{attribute 'GeneratedUsingTerminal: EL9930-0000-0017'}
{attribute addProperty BoxType "EL9930-0000-0017"}
{attribute addProperty Id "A_0004_EL9930_0001_0017EL9930_07FC3A1D4"}
{attribute addProperty CRC "2528476189"}
{attribute addProperty Size "4"}
TYPE A_0003_EL9930_0000_0017_96B57C1D EXTENDS EL9930_B8165E3C :
STRUCT
	{attribute addProperty Name "A_0004_EL9930_0001_0017"}
	{attribute addProperty PreviousPort "A_0003(EL9930-0000-0017) : B"}
	A_0004_EL9930_0001_0017 : EL9930_07FC3A1D;
END_STRUCT
END_TYPE

(* stored: Version 1.2.0.0, ProductVersion 3.1.4024.9
   DUT A_0003_EL9930_0000_0017_96B57C1D: Id {26c4b29d-9ff2-417f-9930-31a4c0fd81f5} *)
